Staubli VAL3: interpolateVel.pgx

program interpolateVel(MotionCmd x_mMotion)
begin
  // Applies velocity "smoothing" to last point in trajectory when vel==0 is replaced by vel==0.1 (default for MoveIt)

  // Round to remove trailing decimal places from fromBinary()
  x_mMotion.mDesc.vel = x_mMotion.mDesc.vel * 10000
  x_mMotion.mDesc.vel = round(x_mMotion.mDesc.vel)
  x_mMotion.mDesc.vel = x_mMotion.mDesc.vel / 10000
  // Smooth last point in traj
  if((x_mMotion.mDesc.vel == 0.1) and (x_mMotion.nSequence != 0))
    x_mMotion.mDesc.vel = (nVel[0] - (nVel[1] - nVel[0]))
  endIf

end
